// TwinCAT 3 PLC project TwinCAT_OPC_UA_Server
// ProgramVersion: 3.1.4023.0
// libraries:
//   Tc2_Standard, * (Beckhoff Automation GmbH)
//   Tc2_System, * (Beckhoff Automation GmbH)
//   Tc3_Module, * (Beckhoff Automation GmbH)
// project tree:
//   GVLs/ OPCUA.TcGVL
//   / PlcTask.TcTTO
//   POUs/ MAIN.TcPOU
// real-time tasks:
//   TASK PlcTask: cycle T#10ms, priority 20, ADS port 350

CONFIGURATION TwinCAT_OPC_UA_Server
    RESOURCE PLC ON TwinCAT3
        TASK PlcTask(INTERVAL := T#10ms, PRIORITY := 20);
        PROGRAM MAIN WITH PlcTask : MAIN;
    END_RESOURCE
END_CONFIGURATION

// ---- GVLs/OPCUA.TcGVL
{attribute 'qualified_only'}
VAR_GLOBAL
	
	{attribute 'OPC.UA.DA' := '1'}
	bBool1:BOOL;
	{attribute 'OPC.UA.DA' := '1'}
	bBool2:BOOL;
	{attribute 'OPC.UA.DA' := '1'}
	bBool3:BOOL;
	
	{attribute 'OPC.UA.DA' := '1'}
	iInt1:INT;
	{attribute 'OPC.UA.DA' := '1'}
	iInt2:INT;
	{attribute 'OPC.UA.DA' := '1'}
	iInt3:INT;
END_VAR

// ---- POUs/MAIN.TcPOU
PROGRAM MAIN
VAR
END_VAR

opcua.bBool1 := opcua.bBool2;
opcua.iInt3 := opcua.iInt1 + opcua.iInt2;

END_PROGRAM
